// Mitsubishi GX Works2 project: PLC_GROUP_04l   PLC: FX3G

// global labels: Global1
VAR_GLOBAL
  StartWorkingDay AT X007 : BOOL;
  Input_Raspberry AT D1100 : INT;
  Input_Lemon AT D1103 : INT;
  Stock_Lemon AT D1111 : INT;
  Input_Stabilizer AT D1105 : INT;
  Stock_Stabilizer AT D1113 : INT;
  Input_GummyBears AT D1107 : INT;
  Stock_GummyBears AT D1115 : INT;
  Lamp AT Y007 : BOOL;
  EmergencyButton AT X005 : BOOL;
  M_NoStock AT M20 : BOOL;
  Storage_Stock AT D1117 : INT;
END_VAR
VAR_GLOBAL CONSTANT
  Reset : INT;
END_VAR
VAR_GLOBAL
  Analog_Display_Value AT D8282 : INT;
  StartPreparation AT X001 : BOOL;
  Analog_Input1 AT D8280 : INT;
END_VAR
VAR_GLOBAL CONSTANT
  TopLimit : INT := 2400;
END_VAR
VAR_GLOBAL
  Regular AT M1 : BOOL;
END_VAR
VAR_GLOBAL CONSTANT
  MinLimit : INT := 2000;
END_VAR
VAR_GLOBAL
  Indulgent AT M2 : BOOL;
END_VAR
VAR_GLOBAL CONSTANT
  Raspberry_Per_Pack : INT;
  Lemon_Per_Unit : INT := 455;
  Stabilizer_Per_Unit : INT := 105;
  GummyBears_Per_Unit : INT := 28;
  Raspberry_Per_Unit : INT := 280;
  Raspberry_Per_Unit_Indulgent : INT := 385;
  Lemon_Per_Unit_Indulgent : INT := 665;
  Stabilizer_Per_Unit_Indulgent : INT := 210;
  GummyBears_Per_Unit_Indulgent : INT := 70;
END_VAR
VAR_GLOBAL
  Start_Regular_Production AT M10 : BOOL;
  Start_Indulgent_Production AT M11 : BOOL;
  Timer_Prep AT TC1 : BOOL;
END_VAR
VAR_GLOBAL CONSTANT
  Prep5 : INT := 50;
END_VAR
VAR_GLOBAL
  FInish_Prep AT TS1 : BOOL;
  PrepProcess AT Y000 : BOOL;
  Timer_Prep_Indulgent AT TC2 : BOOL;
  FInish_Prep_Indulgent AT TS2 : BOOL;
  Tank_Raspberry AT D1123 : INT;
  Tank_Lemon AT D1125 : INT;
  Stock_Raspberry AT D1109 : INT;
  Regular_noStock AT M21 : BOOL;
  Indulgent_noStock AT M22 : BOOL;
  CoolingTransfer AT X002 : BOOL;
  CoolTank_Raspberry AT D1127 : INT;
  CoolTank_Lemon AT D1129 : INT;
  Cooling_State AT M30 : BOOL;
  CoolingProcess AT Y002 : BOOL;
  Timer_Cooling AT TC3 : BOOL;
END_VAR
VAR_GLOBAL CONSTANT
  CoolTime : INT := 80;
END_VAR
VAR_GLOBAL
  TempSensor AT X003 : BOOL;
  FInish_Cooling AT TS3 : BOOL;
  Mixing_State AT M40 : BOOL;
  Timer_Mixing AT TC4 : BOOL;
END_VAR
VAR_GLOBAL CONSTANT
  MixTime_Regular : INT := 30;
END_VAR
VAR_GLOBAL
  Timer_Mixing_Indulgent AT TC5 : BOOL;
END_VAR
VAR_GLOBAL CONSTANT
  MixTime_Idulgent : INT := 50;
END_VAR
VAR_GLOBAL
  Blink_Reset AT M50 : BOOL;
  Timer_Blink1 AT TC6 : BOOL;
END_VAR
VAR_GLOBAL CONSTANT
  BlinkTime : INT := 5;
END_VAR
VAR_GLOBAL
  Finish_Blink1 AT TS6 : BOOL;
  Mixer_Lamp1 AT Y005 : BOOL;
  Timer_Blink2 AT TC7 : BOOL;
  Finish_Blink2 AT TS7 : BOOL;
  Mixer_Lamp2 AT Y006 : BOOL;
  Finish_Mixing AT TS4 : BOOL;
  Finish_Mixing_Indulrent AT TS5 : BOOL;
  Temp_Value AT D1140 : REAL;
  Temp_Value2 AT D1142 : REAL;
END_VAR
VAR_GLOBAL CONSTANT
  MaxLimit_Indulgent : INT := 4000;
END_VAR
VAR_GLOBAL
  Finish_Mixing_Indulgent AT TS5 : BOOL;
END_VAR

// task Task_01 (event TRUE, interval 0, priority 31): POU_01

PROGRAM POU_01
VAR CONSTANT
  Time_Prep : DINT := 5;
END_VAR
(* structured ladder/FBD written out as ST: instructions are called as NAME(EN, inputs, outputs); _pN, _eN, _tN stand for wires *)
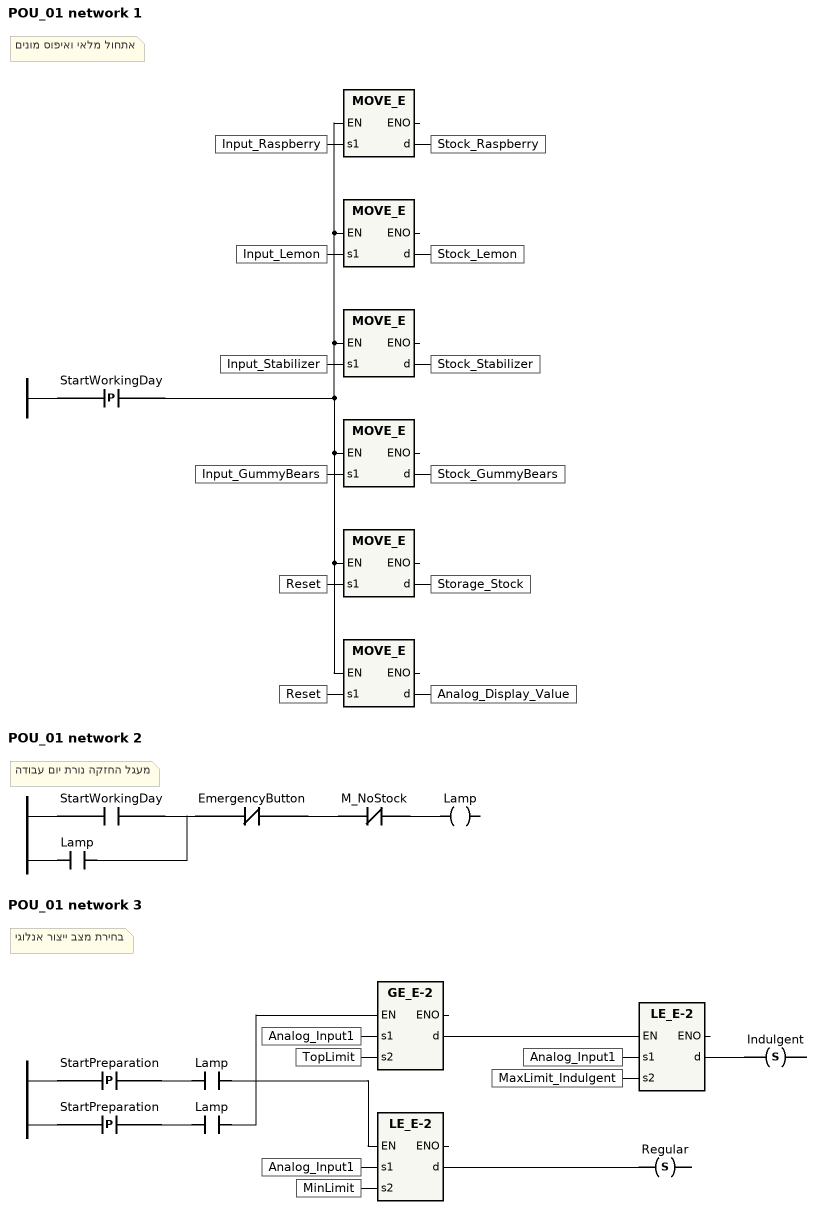
(* network 1 *)
(* אתחול מלאי ואיפוס מונים *)
_p1 := LDP(TRUE, StartWorkingDay);
MOVE_E(_p1, Input_Raspberry, Stock_Raspberry);
MOVE_E(_p1, Input_Lemon, Stock_Lemon);
MOVE_E(_p1, Input_Stabilizer, Stock_Stabilizer);
MOVE_E(_p1, Input_GummyBears, Stock_GummyBears);
MOVE_E(_p1, Reset, Storage_Stock);
MOVE_E(_p1, Reset, Analog_Display_Value);
(* network 2 *)
(* מעגל החזקה נורת יום עבודה *)
Lamp := ((StartWorkingDay OR Lamp) AND NOT EmergencyButton) AND NOT M_NoStock;
(* network 3 *)
(* בחירת מצב ייצור אנלוגי *)
LE_E(LDP(TRUE, StartPreparation) AND Lamp, Analog_Input1, MinLimit, _t1);
SET(_t1, Regular);
GE_E(LDP(TRUE, StartPreparation) AND Lamp, Analog_Input1, TopLimit, _t2);
LE_E(_t2, Analog_Input1, MaxLimit_Indulgent, _t3);
SET(_t3, Indulgent);
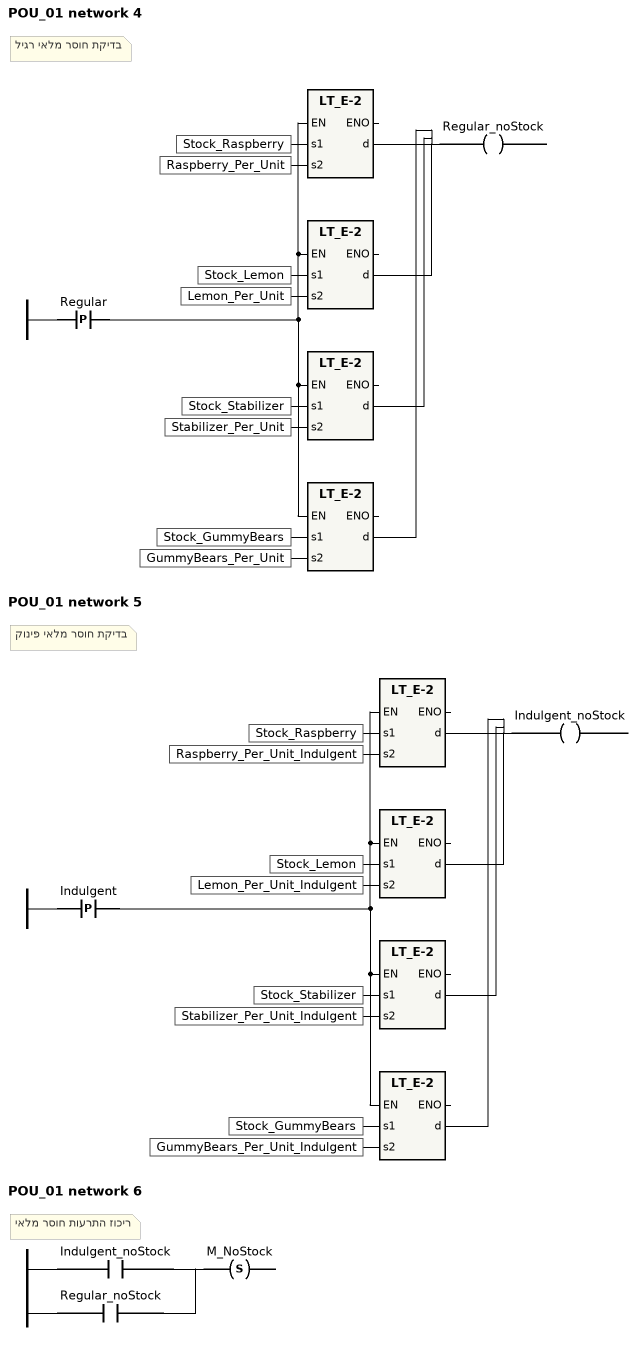
(* network 4 *)
(* בדיקת חוסר מלאי רגיל *)
_p1 := LDP(TRUE, Regular);
LT_E(_p1, Stock_Raspberry, Raspberry_Per_Unit, _t2);
LT_E(_p1, Stock_Lemon, Lemon_Per_Unit, _t3);
LT_E(_p1, Stock_Stabilizer, Stabilizer_Per_Unit, _t4);
LT_E(_p1, Stock_GummyBears, GummyBears_Per_Unit, _t5);
Regular_noStock := _t2 OR _t3 OR _t4 OR _t5;
(* network 5 *)
(* בדיקת חוסר מלאי פינוק *)
_p1 := LDP(TRUE, Indulgent);
LT_E(_p1, Stock_Raspberry, Raspberry_Per_Unit_Indulgent, _t2);
LT_E(_p1, Stock_Lemon, Lemon_Per_Unit_Indulgent, _t3);
LT_E(_p1, Stock_Stabilizer, Stabilizer_Per_Unit_Indulgent, _t4);
LT_E(_p1, Stock_GummyBears, GummyBears_Per_Unit_Indulgent, _t5);
Indulgent_noStock := _t2 OR _t3 OR _t4 OR _t5;
(* network 6 *)
(* ריכוז התרעות חוסר מלאי *)
SET(Indulgent_noStock OR Regular_noStock, M_NoStock);
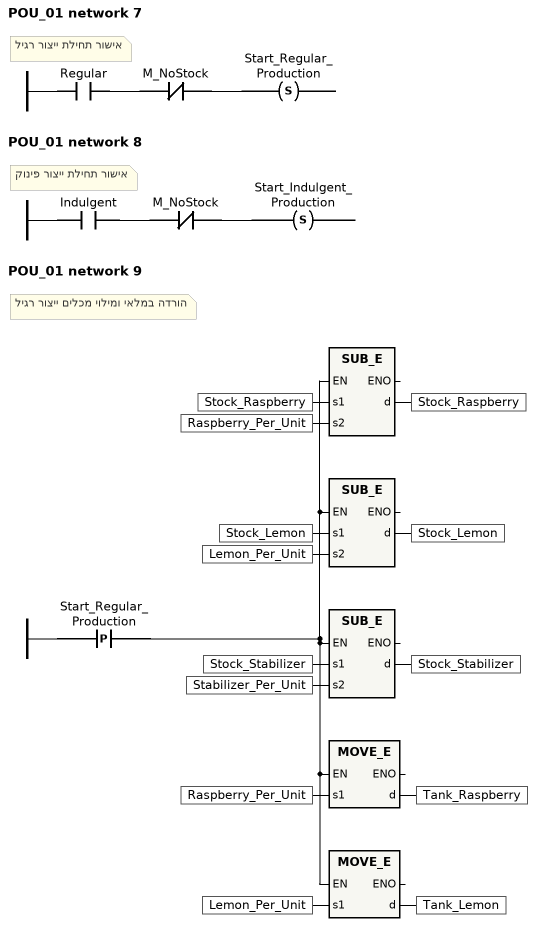
(* network 7 *)
(* אישור תחילת ייצור רגיל *)
SET(Regular AND NOT M_NoStock, Start_Regular_Production);
(* network 8 *)
(* אישור תחילת ייצור פינוק *)
SET(Indulgent AND NOT M_NoStock, Start_Indulgent_Production);
(* network 9 *)
(* הורדה במלאי ומילוי מכלים ייצור רגיל *)
_p1 := LDP(TRUE, Start_Regular_Production);
SUB_E(_p1, Stock_Raspberry, Raspberry_Per_Unit, Stock_Raspberry);
SUB_E(_p1, Stock_Lemon, Lemon_Per_Unit, Stock_Lemon);
SUB_E(_p1, Stock_Stabilizer, Stabilizer_Per_Unit, Stock_Stabilizer);
MOVE_E(_p1, Raspberry_Per_Unit, Tank_Raspberry);
MOVE_E(_p1, Lemon_Per_Unit, Tank_Lemon);
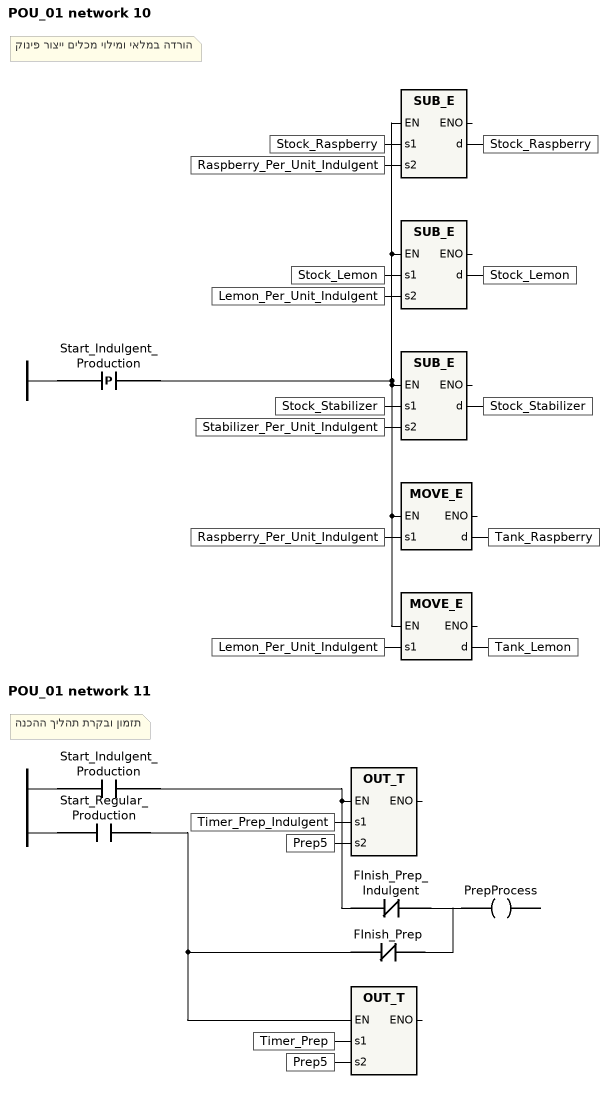
(* network 10 *)
(* הורדה במלאי ומילוי מכלים ייצור פינוק *)
_p1 := LDP(TRUE, Start_Indulgent_Production);
SUB_E(_p1, Stock_Raspberry, Raspberry_Per_Unit_Indulgent, Stock_Raspberry);
SUB_E(_p1, Stock_Lemon, Lemon_Per_Unit_Indulgent, Stock_Lemon);
SUB_E(_p1, Stock_Stabilizer, Stabilizer_Per_Unit_Indulgent, Stock_Stabilizer);
MOVE_E(_p1, Raspberry_Per_Unit_Indulgent, Tank_Raspberry);
MOVE_E(_p1, Lemon_Per_Unit_Indulgent, Tank_Lemon);
(* network 11 *)
(* תזמון ובקרת תהליך ההכנה *)
OUT_T(Start_Indulgent_Production, Timer_Prep_Indulgent, Prep5);
PrepProcess := (Start_Indulgent_Production AND NOT FInish_Prep_Indulgent) OR (Start_Regular_Production AND NOT FInish_Prep);
OUT_T(Start_Regular_Production, Timer_Prep, Prep5);
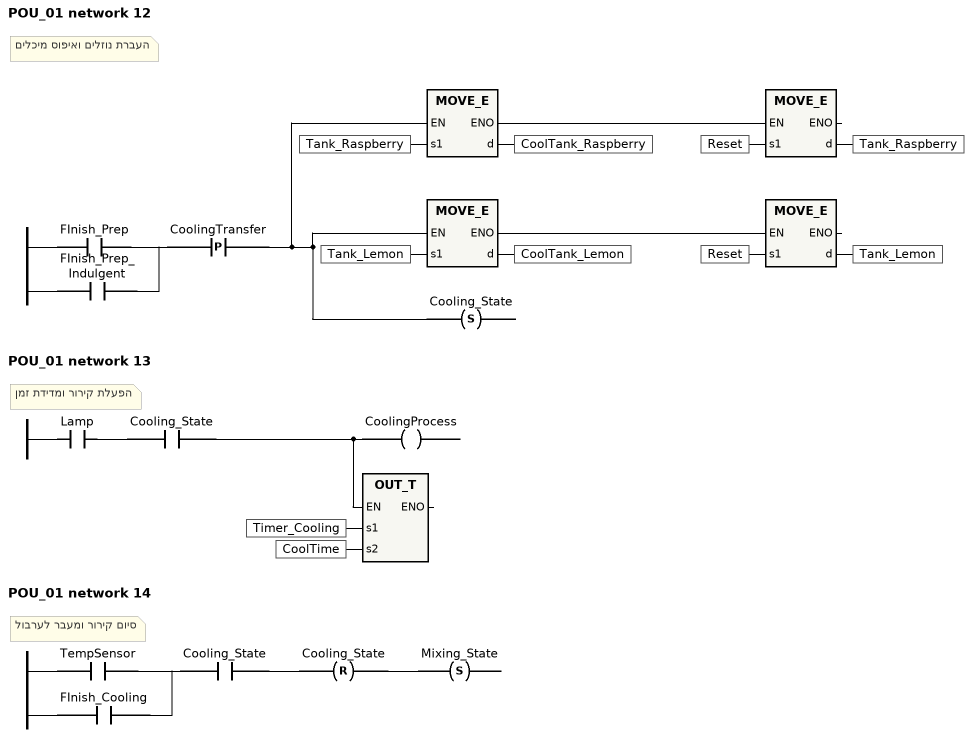
(* network 12 *)
(* העברת נוזלים ואיפוס מיכלים *)
_p1 := (FInish_Prep OR FInish_Prep_Indulgent) AND LDP(TRUE, CoolingTransfer);
_e2 := MOVE_E(_p1, Tank_Raspberry, CoolTank_Raspberry);
MOVE_E(_e2, Reset, Tank_Raspberry);
_e3 := MOVE_E(_p1, Tank_Lemon, CoolTank_Lemon);
MOVE_E(_e3, Reset, Tank_Lemon);
SET(_p1, Cooling_State);
(* network 13 *)
(* הפעלת קירור ומדידת זמן *)
_p1 := Lamp AND Cooling_State;
CoolingProcess := _p1;
OUT_T(_p1, Timer_Cooling, CoolTime);
(* network 14 *)
(* סיום קירור ומעבר לערבול *)
_p1 := (TempSensor OR FInish_Cooling) AND Cooling_State;
RST(_p1, Cooling_State);
SET(_p1, Mixing_State);
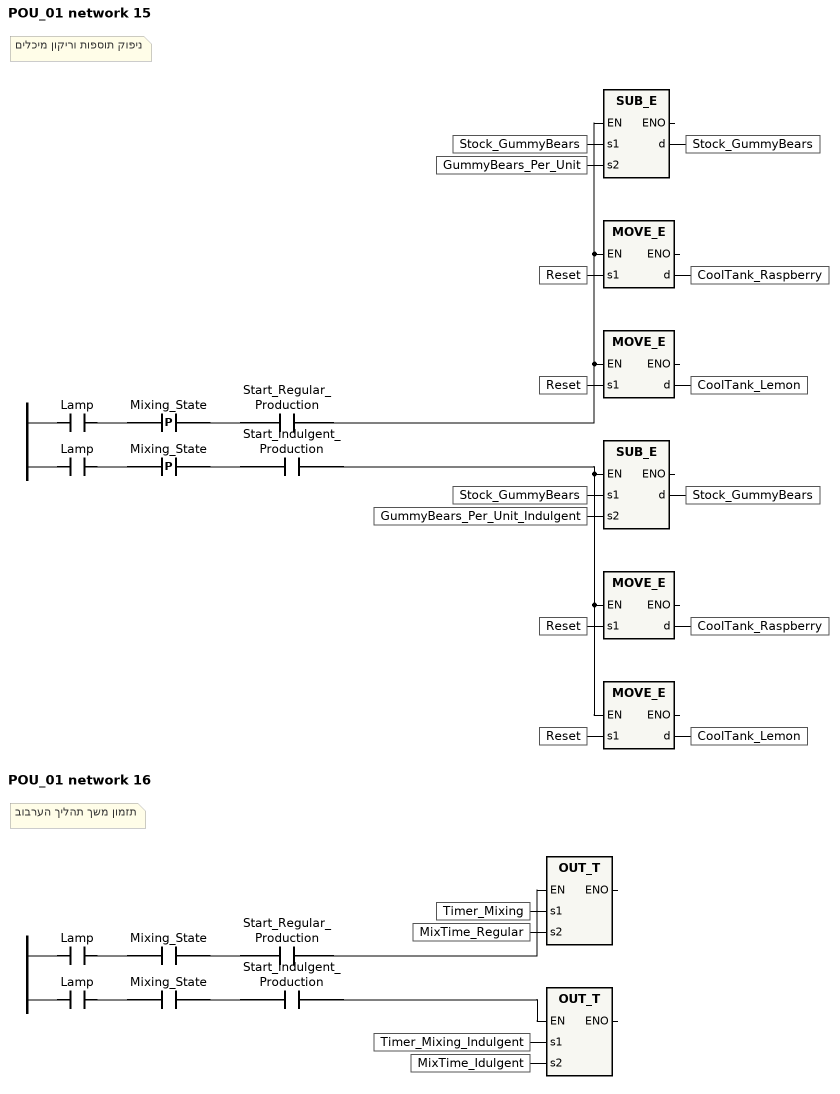
(* network 15 *)
(* ניפוק תוספות וריקון מיכלים *)
_p1 := Lamp AND LDP(TRUE, Mixing_State) AND Start_Regular_Production;
SUB_E(_p1, Stock_GummyBears, GummyBears_Per_Unit, Stock_GummyBears);
MOVE_E(_p1, Reset, CoolTank_Raspberry);
MOVE_E(_p1, Reset, CoolTank_Lemon);
_p2 := Lamp AND LDP(TRUE, Mixing_State) AND Start_Indulgent_Production;
SUB_E(_p2, Stock_GummyBears, GummyBears_Per_Unit_Indulgent, Stock_GummyBears);
MOVE_E(_p2, Reset, CoolTank_Raspberry);
MOVE_E(_p2, Reset, CoolTank_Lemon);
(* network 16 *)
(* תזמון משך תהליך הערבוב *)
OUT_T(Lamp AND Mixing_State AND Start_Regular_Production, Timer_Mixing, MixTime_Regular);
OUT_T(Lamp AND Mixing_State AND Start_Indulgent_Production, Timer_Mixing_Indulgent, MixTime_Idulgent);
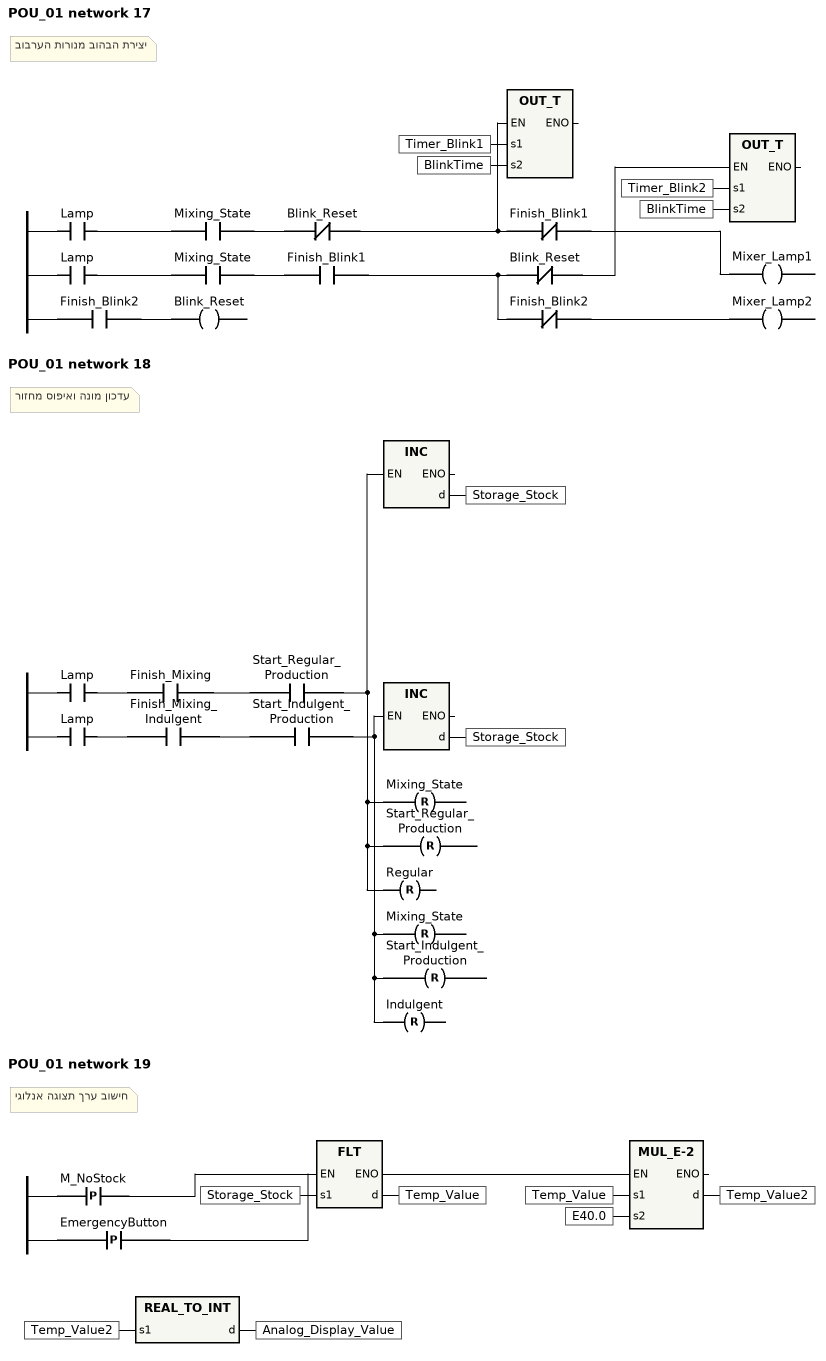
(* network 17 *)
(* יצירת הבהוב מנורות הערבוב *)
_p1 := Lamp AND Mixing_State AND NOT Blink_Reset;
OUT_T(_p1, Timer_Blink1, BlinkTime);
Mixer_Lamp1 := _p1 AND NOT Finish_Blink1;
_p2 := Lamp AND Mixing_State AND Finish_Blink1;
OUT_T(_p2 AND NOT Blink_Reset, Timer_Blink2, BlinkTime);
Mixer_Lamp2 := _p2 AND NOT Finish_Blink2;
Blink_Reset := Finish_Blink2;
(* network 18 *)
(* עדכון מונה ואיפוס מחזור *)
_p1 := Lamp AND Finish_Mixing AND Start_Regular_Production;
INC(_p1, Storage_Stock);
RST(_p1, Mixing_State);
RST(_p1, Start_Regular_Production);
RST(_p1, Regular);
_p2 := Lamp AND Finish_Mixing_Indulgent AND Start_Indulgent_Production;
INC(_p2, Storage_Stock);
RST(_p2, Mixing_State);
RST(_p2, Start_Indulgent_Production);
RST(_p2, Indulgent);
(* network 19 *)
(* חישוב ערך תצוגה אנלוגי *)
Analog_Display_Value := REAL_TO_INT(Temp_Value2);
_e1 := FLT(LDP(TRUE, M_NoStock) OR LDP(TRUE, EmergencyButton), Storage_Stock, Temp_Value);
MUL_E(_e1, Temp_Value, E40.0, Temp_Value2);
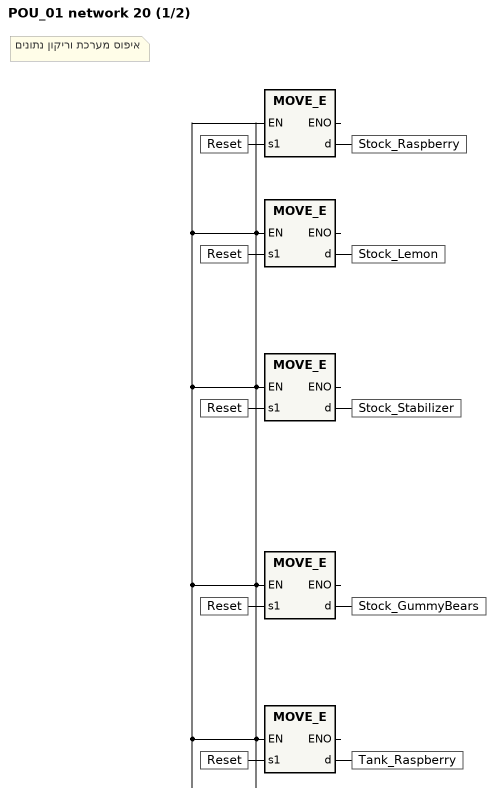
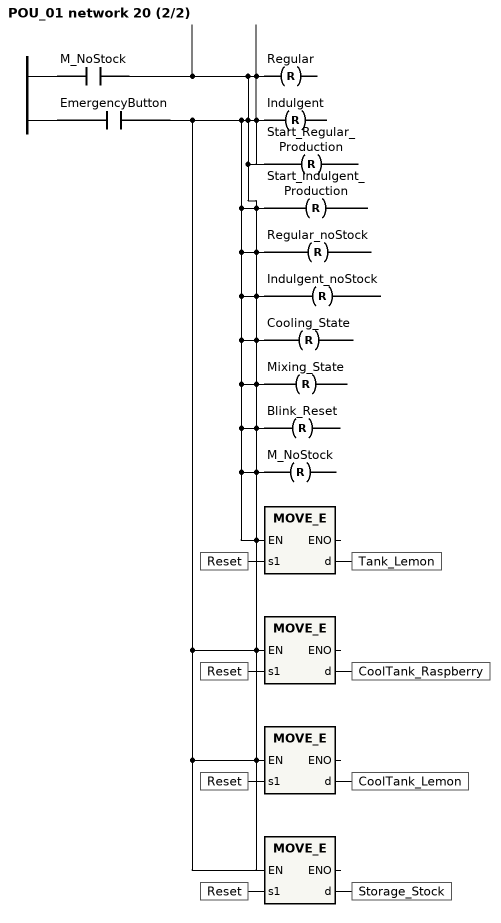
(* network 20 *)
(* איפוס מערכת וריקון נתונים *)
_p1 := M_NoStock OR EmergencyButton;
MOVE_E(_p1, Reset, Stock_Raspberry);
MOVE_E(_p1, Reset, Stock_Lemon);
RST(_p1, Regular);
RST(_p1, Indulgent);
MOVE_E(_p1, Reset, Stock_Stabilizer);
RST(_p1, Start_Regular_Production);
MOVE_E(_p1, Reset, Stock_GummyBears);
RST(_p1, Start_Indulgent_Production);
MOVE_E(_p1, Reset, Tank_Raspberry);
RST(_p1, Regular_noStock);
RST(_p1, Indulgent_noStock);
MOVE_E(_p1, Reset, Tank_Lemon);
RST(_p1, Cooling_State);
MOVE_E(_p1, Reset, CoolTank_Raspberry);
RST(_p1, Mixing_State);
MOVE_E(_p1, Reset, CoolTank_Lemon);
RST(_p1, Blink_Reset);
RST(_p1, M_NoStock);
MOVE_E(_p1, Reset, Storage_Stock);
END_PROGRAM
